FUNCTION_BLOCK POU EXTENDS AxisBase
VAR_INPUT
END_VAR
VAR_OUTPUT
END_VAR
VAR
END_VAR

END_FUNCTION_BLOCK

(* stored: Version 1.1.0.1, ProductVersion 3.1.4024.12
   POU POU: Id {d16e7e0b-bbc7-44ae-945d-c3117fa5342e}, SpecialFunc None *)
